Fanuc KAREL source: kt00021.KL

PROGRAM KT00021
%NOLOCKGROUP
VAR
Y1 : ARRAY[2] OF BYTE
Y2 : ARRAY[2] OF BYTE
OUT:INTEGER
BEGIN
Y1[1]=2
Y2[1]=3
Y1[1]=2
Y2[1]=3
OUT=(Y1[1] + Y2[1])
END KT00021
